INTERFACE I_Subscriber

METHOD update : BOOL
VAR_INPUT
	in_sContent			: STRING;
END_VAR
END_METHOD

END_INTERFACE

(* stored: Version 1.1.0.1
   Itf I_Subscriber: Id {3f63c4dc-1a6a-4f91-8756-8a38f183caeb}
   Method update: Id {0e8c22c7-2307-4396-afc8-1a0a21b53673} *)
